{attribute 'GeneratedUsingTerminal: EPP1321-0060-0016'}
{attribute addProperty BoxType "EPP1321-0060-0016"}
{attribute addProperty Id "A_0019_EPP1322_0001_0016A_0019_EPP1322_0001_0016_88121AEB322"}
{attribute addProperty CRC "3809713363"}
{attribute addProperty Size "322"}
TYPE A_0018_EPP1321_0060_0016_E3139CD3 EXTENDS EPP1321_1FC0878B :
STRUCT
	{attribute addProperty Name "A_0019_EPP1322_0001_0016"}
	{attribute addProperty PreviousPort "A_0018(EPP1321-0060-0016) : D"}
	A_0019_EPP1322_0001_0016 : A_0019_EPP1322_0001_0016_88121AEB;
END_STRUCT
END_TYPE

(* stored: Version 1.2.0.0, ProductVersion 3.1.4024.9
   DUT A_0018_EPP1321_0060_0016_E3139CD3: Id {724a851c-16dd-4b12-a479-a50de5b7a30d} *)
